// TIA Portal V21 export
DATA_BLOCK "BatchDetailsLength_DB"   // DB40
// stored: InstanceOfName BatchDetailsLength, InstanceOfType FB
"BatchDetailsLength"
   // VAR_OUTPUT
   //    EquipmentID_Len { ExternalAccessible := 'False'; ExternalVisible := 'False'; ExternalWritable := 'False'} : Int;
   //    ProductName_Len { ExternalAccessible := 'False'; ExternalVisible := 'False'; ExternalWritable := 'False'} : Int;
   //    BatchNum_Len { ExternalAccessible := 'False'; ExternalVisible := 'False'; ExternalWritable := 'False'} : Int;
   //    PrintInt_Len { ExternalAccessible := 'False'; ExternalVisible := 'False'; ExternalWritable := 'False'} : Int;
   // END_VAR
BEGIN
END_DATA_BLOCK
